FUNCTION_BLOCK HaltMoverTask_TestSuite
VAR
	stubAxis : AXIS_REF;
	testHaltMover : HaltMoverTask := (AxisRef := stubAxis);
	ThisTestSuite : TestSuite<TestSuiteParameter.MaxTestCount>('C:\ProgramData\Beckhoff\TwinCAT\3.1\Boot\HaltMover_Tests.xml') := (TestSuiteName := 'HaltMover Test Suite');
END_VAR

TaskRejectsCommandWithNoAxisRef_Test();
TaskRejectsDuplicateCommand_Test();
TaskWontCycleWithoutAxisRef_Test();
TaskAcceptsCommand_Test();
TaskRejectsZeroDecel_Test();
TaskRejectsZeroJerk_Test();
TaskRejectsInvalidGap_Test();

METHOD TaskAcceptsCommand_Test
VAR_INST
	Expected : BOOL := TRUE;
	Actual	 : BOOL;
END_VAR
IF ThisTestSuite.Test(__POUNAME()).ExecuteTest() THEN
	Actual := Succeeded(testHaltMover.Execute());
	testHaltMover.Abort();
	ThisTestSuite.Test(__POUNAME()).AssertEqual(Expected, Actual);
END_IF
END_METHOD

METHOD TaskRejectsCommandWithNoAxisRef_Test
VAR_INST
	Expected : BOOL := TRUE;
	Actual	 : BOOL;
END_VAR
IF ThisTestSuite.Test(__POUNAME()).ExecuteTest() THEN
	testHaltMover.AxisRef REF= 16#0;
	Actual := FAILED(testHaltMover.Execute());
	testHaltMover.Abort();
	testHaltMover.AxisRef REF= stubAxis;
	ThisTestSuite.Test(__POUNAME()).AssertEqual(Expected, Actual);
END_IF
END_METHOD

METHOD TaskRejectsDuplicateCommand_Test
VAR_INST
	Expected : BOOL := TRUE;
	Actual	 : BOOL;
END_VAR
IF ThisTestSuite.Test(__POUNAME()).ExecuteTest() THEN
	testHaltMover.Execute();
	Actual := FAILED(testHaltMover.Execute());
	testHaltMover.Abort();
	ThisTestSuite.Test(__POUNAME()).AssertEqual(Expected, Actual);
END_IF
END_METHOD

METHOD TaskRejectsInvalidGap_Test
VAR_INST
	Expected : BOOL := TRUE;
	Actual	 : BOOL;
END_VAR
IF ThisTestSuite.Test(__POUNAME()).ExecuteTest() THEN
	testHaltMover.Gap := 1000.0;
	testHaltMover.Gap := 25.0;
	Actual := testHaltMover.Jerk > 50.0;
	ThisTestSuite.Test(__POUNAME()).AssertEqual(Expected, Actual);
END_IF
END_METHOD

METHOD TaskRejectsZeroDecel_Test
VAR_INST
	Expected : BOOL := TRUE;
	Actual	 : BOOL;
END_VAR
IF ThisTestSuite.Test(__POUNAME()).ExecuteTest() THEN
	testHaltMover.Deceleration := 1000.0;
	testHaltMover.Deceleration := 0.0;
	Actual := testHaltMover.Deceleration <> 0.0;
	ThisTestSuite.Test(__POUNAME()).AssertEqual(Expected, Actual);
END_IF
END_METHOD

METHOD TaskRejectsZeroJerk_Test
VAR_INST
	Expected : BOOL := TRUE;
	Actual	 : BOOL;
END_VAR
IF ThisTestSuite.Test(__POUNAME()).ExecuteTest() THEN
	testHaltMover.Jerk := 1000.0;
	testHaltMover.Jerk := 0.0;
	Actual := testHaltMover.Jerk <> 0.0;
	ThisTestSuite.Test(__POUNAME()).AssertEqual(Expected, Actual);
END_IF
END_METHOD

METHOD TaskWontCycleWithoutAxisRef_Test
VAR_INST
	Expected : BOOL := TRUE;
	Actual	 : BOOL;
END_VAR
IF ThisTestSuite.Test(__POUNAME()).ExecuteTest() THEN
	testHaltMover.AxisRef REF= 16#0;
	Actual := FAILED(testHaltMover.Cycle());
	testHaltMover.Abort();
	testHaltMover.AxisRef REF= stubAxis;
	ThisTestSuite.Test(__POUNAME()).AssertEqual(Expected, Actual);
END_IF
END_METHOD

END_FUNCTION_BLOCK

(* stored: Version 1.1.0.1
   POU HaltMoverTask_TestSuite: Id {d7b1227a-089d-4d2d-9759-410675fe30bc}, SpecialFunc None
   Method TaskAcceptsCommand_Test: Id {fb6fb1d2-beaf-43e9-a2b1-bb05d4d56bf2}
   Method TaskRejectsCommandWithNoAxisRef_Test: Id {78fc3f65-b7dc-45a5-8cf9-915543da9eb3}
   Method TaskRejectsDuplicateCommand_Test: Id {bd7d62a4-1b55-4518-ac05-e7232036c5c4}
   Method TaskRejectsInvalidGap_Test: Id {3fbde906-4c70-4bb7-b8a4-fe505520d990}
   Method TaskRejectsZeroDecel_Test: Id {6e7b6622-a53d-4b78-9592-e7b8fdc3d9ea}
   Method TaskRejectsZeroJerk_Test: Id {398c4671-f64c-4f24-abfa-aad4dea4b2a1}
   Method TaskWontCycleWithoutAxisRef_Test: Id {936e1fe3-a6d5-43d7-8093-3d608f36ee71} *)
